% RSLogix 500 project PROJECT3_INVENTORY_MANAGEMENT.RSS, saved by version 8.30.00.16 %
PROJECT "UNTITLED"    % processor: Bul.1763 MicroLogix 1100 Series B %

PROGRAM FILES
  LAD 2   14 rungs

DATA FILES
  O0 OUTPUT  4 elements
  I1 INPUT  6 elements
  S2 STATUS  66 elements
  B3 BINARY  1 elements
  T4 TIMER  1 elements
  C5 COUNTER  1 elements
  R6 CONTROL  1 elements
  N7 INTEGER  10 elements
  F8 FLOAT  1 elements
  ST9 BARCODE  13 elements

LADDER 2
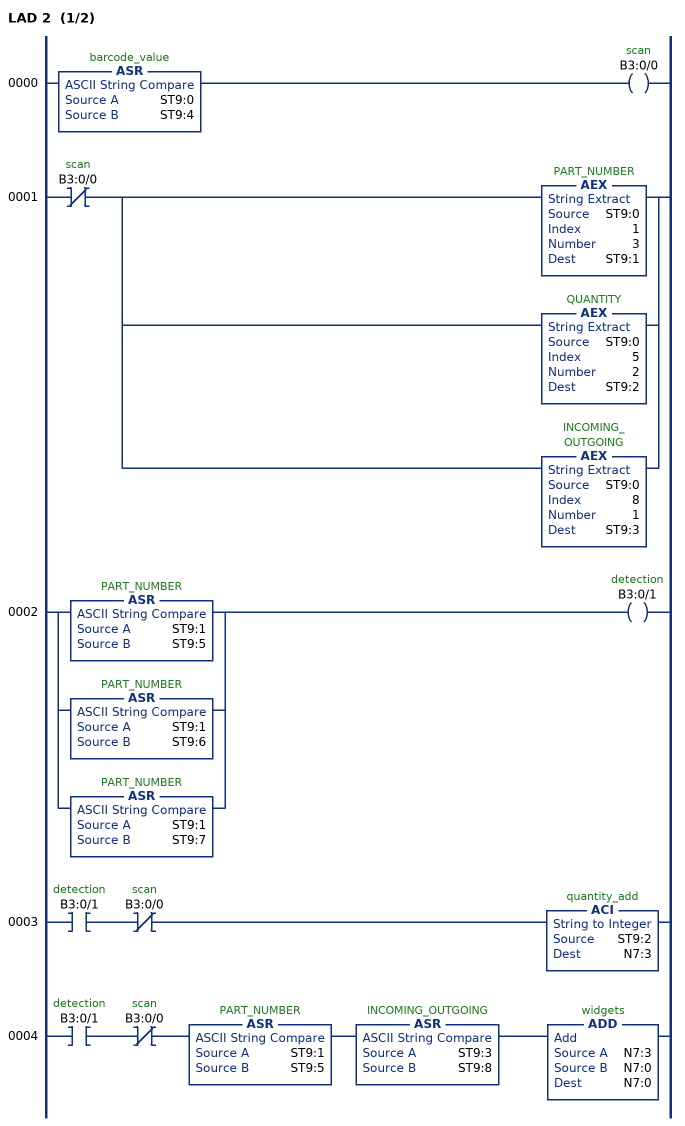
% Rung: 0 %
SOR ASR ST9:0 ST9:4 OTE B3:0/0 EOR
%   ST9:0  "barcode_value" %
%   ST9:4  "value" %
%   B3:0/0  "scan" %
% Rung: 1 %
SOR XIO B3:0/0 BST AEX ST9:0 1 3 ST9:1 NXB AEX ST9:0 5 2 ST9:2 NXB AEX ST9:0 8 1 ST9:3 BND EOR
%   B3:0/0  "scan" %
%   ST9:0  "barcode_value" %
%   ST9:1  PART_NUMBER %
%   ST9:2  QUANTITY %
%   ST9:3  INCOMING_OUTGOING %
% Rung: 2 %
SOR BST ASR ST9:1 ST9:5 NXB ASR ST9:1 ST9:6 NXB ASR ST9:1 ST9:7 BND OTE B3:0/1 EOR
%   ST9:1  PART_NUMBER %
%   ST9:5  "widgets" %
%   ST9:6  "doodads" %
%   ST9:7  "wockies" %
%   B3:0/1  "detection" %
% Rung: 3 %
SOR XIC B3:0/1 XIO B3:0/0 ACI ST9:2 N7:3 EOR
%   B3:0/1  "detection" %
%   B3:0/0  "scan" %
%   ST9:2  QUANTITY %
%   N7:3  "quantity_add" %
% Rung: 4 %
SOR XIC B3:0/1 XIO B3:0/0 ASR ST9:1 ST9:5 ASR ST9:3 ST9:8 ADD N7:3 N7:0 N7:0 EOR
%   B3:0/1  "detection" %
%   B3:0/0  "scan" %
%   ST9:1  PART_NUMBER %
%   ST9:5  "widgets" %
%   ST9:3  INCOMING_OUTGOING %
%   ST9:8  "1" %
%   N7:3  "quantity_add" %
%   N7:0  "widgets" %

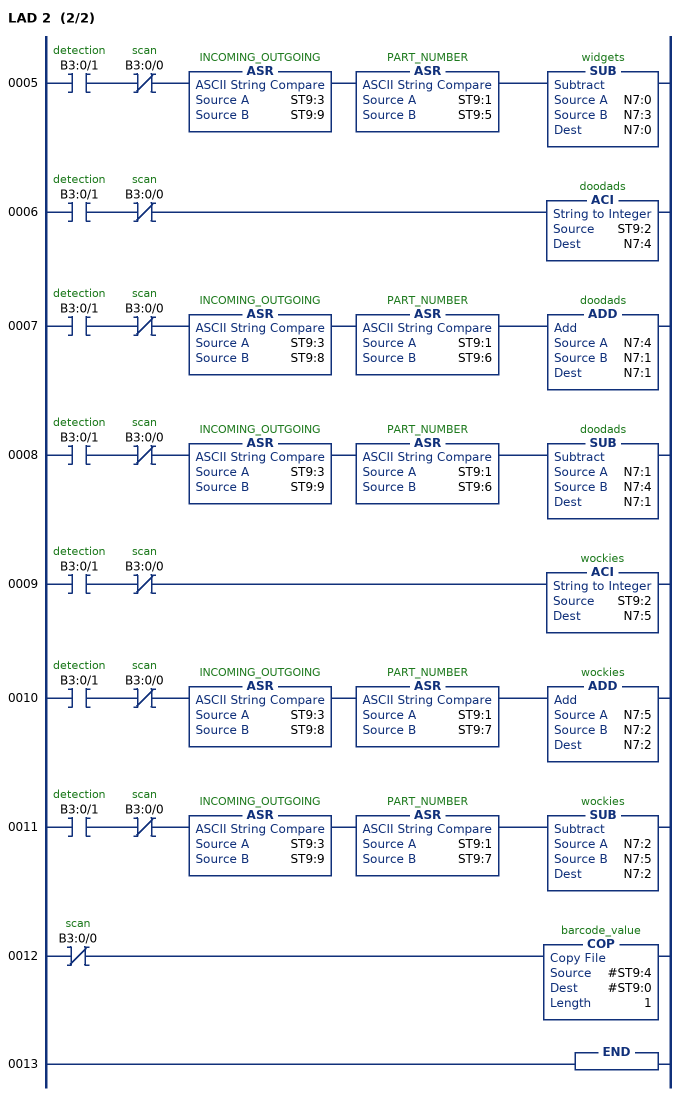
% Rung: 5 %
SOR XIC B3:0/1 XIO B3:0/0 ASR ST9:3 ST9:9 ASR ST9:1 ST9:5 SUB N7:0 N7:3 N7:0 EOR
%   B3:0/1  "detection" %
%   B3:0/0  "scan" %
%   ST9:3  INCOMING_OUTGOING %
%   ST9:9  "2" %
%   ST9:1  PART_NUMBER %
%   ST9:5  "widgets" %
%   N7:0  "widgets" %
%   N7:3  "quantity_add" %
% Rung: 6 %
SOR XIC B3:0/1 XIO B3:0/0 ACI ST9:2 N7:4 EOR
%   B3:0/1  "detection" %
%   B3:0/0  "scan" %
%   ST9:2  QUANTITY %
%   N7:4  "doodads" %
% Rung: 7 %
SOR XIC B3:0/1 XIO B3:0/0 ASR ST9:3 ST9:8 ASR ST9:1 ST9:6 ADD N7:4 N7:1 N7:1 EOR
%   B3:0/1  "detection" %
%   B3:0/0  "scan" %
%   ST9:3  INCOMING_OUTGOING %
%   ST9:8  "1" %
%   ST9:1  PART_NUMBER %
%   ST9:6  "doodads" %
%   N7:4  "doodads" %
%   N7:1  "doodads" %
% Rung: 8 %
SOR XIC B3:0/1 XIO B3:0/0 ASR ST9:3 ST9:9 ASR ST9:1 ST9:6 SUB N7:1 N7:4 N7:1 EOR
%   B3:0/1  "detection" %
%   B3:0/0  "scan" %
%   ST9:3  INCOMING_OUTGOING %
%   ST9:9  "2" %
%   ST9:1  PART_NUMBER %
%   ST9:6  "doodads" %
%   N7:1  "doodads" %
%   N7:4  "doodads" %
% Rung: 9 %
SOR XIC B3:0/1 XIO B3:0/0 ACI ST9:2 N7:5 EOR
%   B3:0/1  "detection" %
%   B3:0/0  "scan" %
%   ST9:2  QUANTITY %
%   N7:5  "wockies" %
% Rung: 10 %
SOR XIC B3:0/1 XIO B3:0/0 ASR ST9:3 ST9:8 ASR ST9:1 ST9:7 ADD N7:5 N7:2 N7:2 EOR
%   B3:0/1  "detection" %
%   B3:0/0  "scan" %
%   ST9:3  INCOMING_OUTGOING %
%   ST9:8  "1" %
%   ST9:1  PART_NUMBER %
%   ST9:7  "wockies" %
%   N7:5  "wockies" %
%   N7:2  "wockies" %
% Rung: 11 %
SOR XIC B3:0/1 XIO B3:0/0 ASR ST9:3 ST9:9 ASR ST9:1 ST9:7 SUB N7:2 N7:5 N7:2 EOR
%   B3:0/1  "detection" %
%   B3:0/0  "scan" %
%   ST9:3  INCOMING_OUTGOING %
%   ST9:9  "2" %
%   ST9:1  PART_NUMBER %
%   ST9:7  "wockies" %
%   N7:2  "wockies" %
%   N7:5  "wockies" %
% Rung: 12 %
SOR XIO B3:0/0 COP #ST9:4 #ST9:0 1 EOR
%   B3:0/0  "scan" %
%   ST9:4  "value" %
%   ST9:0  "barcode_value" %
% Rung: 13 %
SOR END EOR

OTHER DOCUMENTED ADDRESSES
  N7:7  "wid"
  N7:8  "doo"
  N7:9  "wock"
  ST9:10  "widgets_store"
  ST9:10.0  "widgets_store_capaci ty"
  ST9:11  "Doodads_store_capaci ty"
  ST9:12  "wockies_store"
  ST9:12.0  "wockies_store_capaci ty"

DATA TABLE (non-zero values as saved)
DATA ST9
% ST9:5 % "123"
% ST9:6 % "456"
% ST9:7 % "789"
% ST9:8 % "1"
% ST9:9 % "2"
